PROGRAM MAIN
VAR
END_VAR

END_PROGRAM

(* stored: Version 1.1.0.1
   POU MAIN: Id {0ca768b3-8d21-41b8-97a6-a0ef6f8b0341} *)
